// SIMATIC S7-200 project (STEP 7-Micro/WIN), CPU 224 REL 02.01

ORGANIZATION_BLOCK Briquette_Press_B_40:OB1
TITLE=B V4.0
// Custom program for WEIMA TH Standard Series briquette press.
//  #NVJOB Nicholas Veselov (independent developer) - https://nvjob.pro, http://nvjob.dx.am
// 
// ---------------------------------------------------------------------
// 
// INPUTS
// I0.0 - Power.
// I0.1 - Start the program in automatic mode.
// I0.2 - Stop the program in automatic mode.
// I0.3 - Manual mode.
// I0.4 - Vertical piston, sensor, lower position.
// I0.5 - Vertical piston, sensor, upper position.
// I0.6 - Horizontal piston, sensor, position retracted.
// I0.7 - Horizontal piston, sensor, position extended.
// I1.0 - Not involved.
// I1.1 - Valve button.
// I1.2 - Accident, stop.
// I1.3 - Change in operating time of the screw. Min time*.
// I1.4 - Change in the operating time of the screw. Max. time*.
// I1.5 - Not involved.
// 
// ---------------------------------------------------------------------
// 
// OUTPUTS
// Q0.0 - The engine of the hydraulic power station (star-delta).
// Q0.1 - Hydroelectric power station engine (star-delta).
// Q0.2 - Fan.
// Q0.3 - Auger.
// Q0.4 - Vertical piston, valve, up position (pushes down).
// Q0.5 - Vertical piston, valve, lower position (pushes up).
// Q0.6 - Horizontal piston, valve, retracts the piston.
// Q0.7 - Horizontal piston, valve, extends the piston.
// Q1.0 - Collet Piston.
// Q1.1 - Light Bulb Start
// 
BEGIN
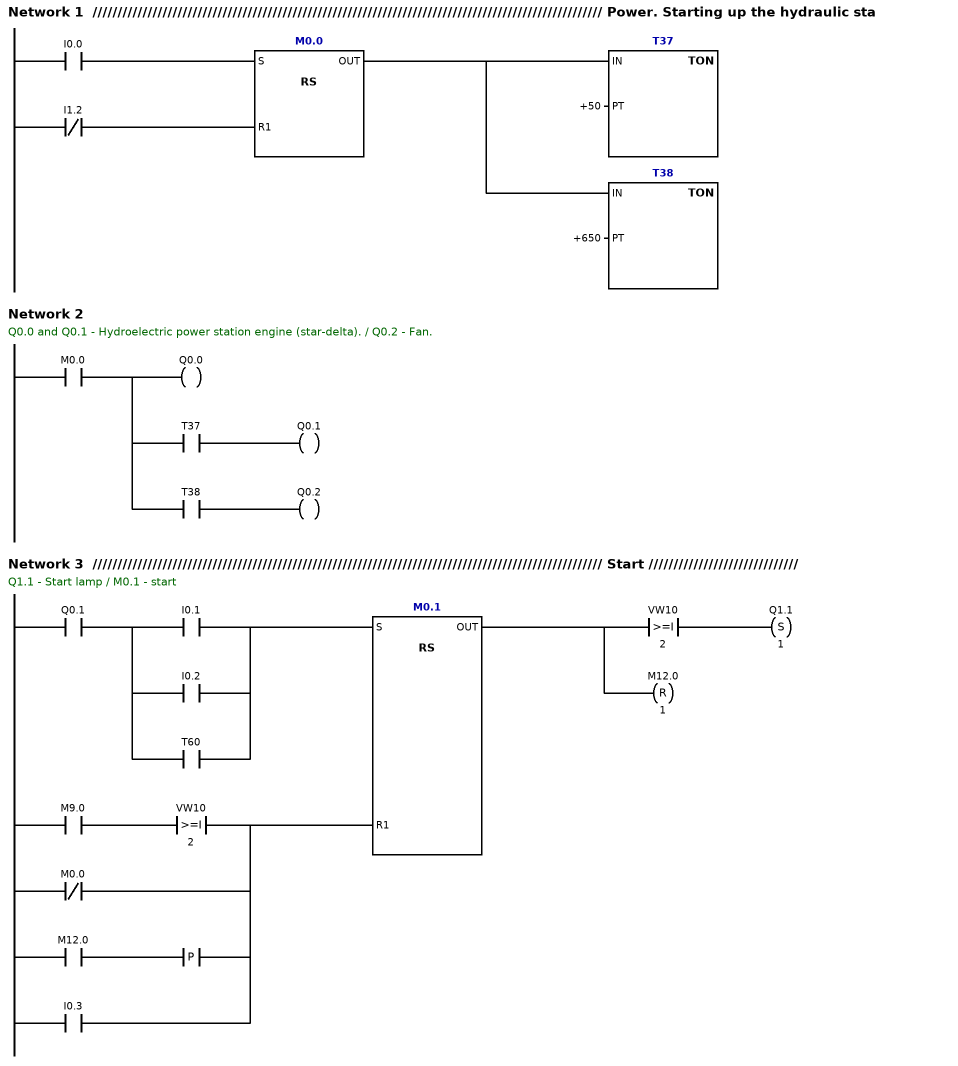
Network 1 // //////////////////////////////////////////////////////////////////////////////////////////////////////
Power. Starting up the hydraulic station.
//////////////////////////////////////////////////////////////////////////////////////////////////////
LD     I0.0
LDN    I1.2
NOT
LPS
A      M0.0
=      M0.0
LPP
ALD
O      M0.0
=      M0.0
TON    T37, +50
TON    T38, +650
Network 2
// Q0.0 and Q0.1 - Hydroelectric power station engine (star-delta).
// Q0.2 - Fan.
LD     M0.0
LPS
=      Q0.0
A      T37
=      Q0.1
LPP
A      T38
=      Q0.2
Network 3 // //////////////////////////////////////////////////////////////////////////////////////////////////////
Start
//////////////////////////////////////////////////////////////////////////////////////////////////////
// Q1.1 - Start lamp
// M0.1 - start
LD     Q0.1
LD     I0.1
O      I0.2
O      T60
ALD
LD     M9.0
AW>=   VW10, 2
ON     M0.0
LD     M12.0
EU
OLD
O      I0.3
NOT
LPS
A      M0.1
=      M0.1
LPP
ALD
O      M0.1
=      M0.1
LPS
AW>=   VW10, 2
S      Q1.1, 1
LPP
R      M12.0, 1
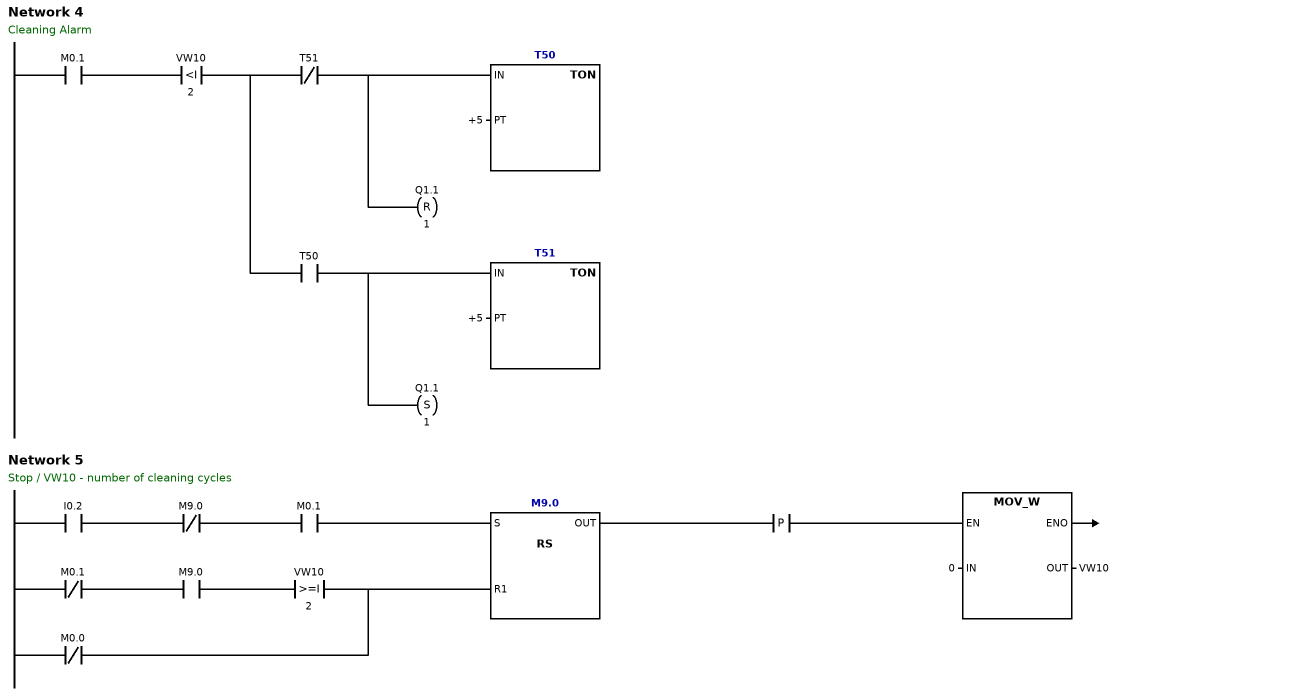
Network 4
// Cleaning Alarm
LD     M0.1
AW<    VW10, 2
LPS
AN     T51
TON    T50, +5
R      Q1.1, 1
LPP
A      T50
TON    T51, +5
S      Q1.1, 1
Network 5
// Stop
// VW10 - number of cleaning cycles
LD     I0.2
AN     M9.0
A      M0.1
LDN    M0.1
A      M9.0
AW>=   VW10, 2
ON     M0.0
NOT
LPS
A      M9.0
=      M9.0
LPP
ALD
O      M9.0
=      M9.0
EU
MOVW   0, VW10
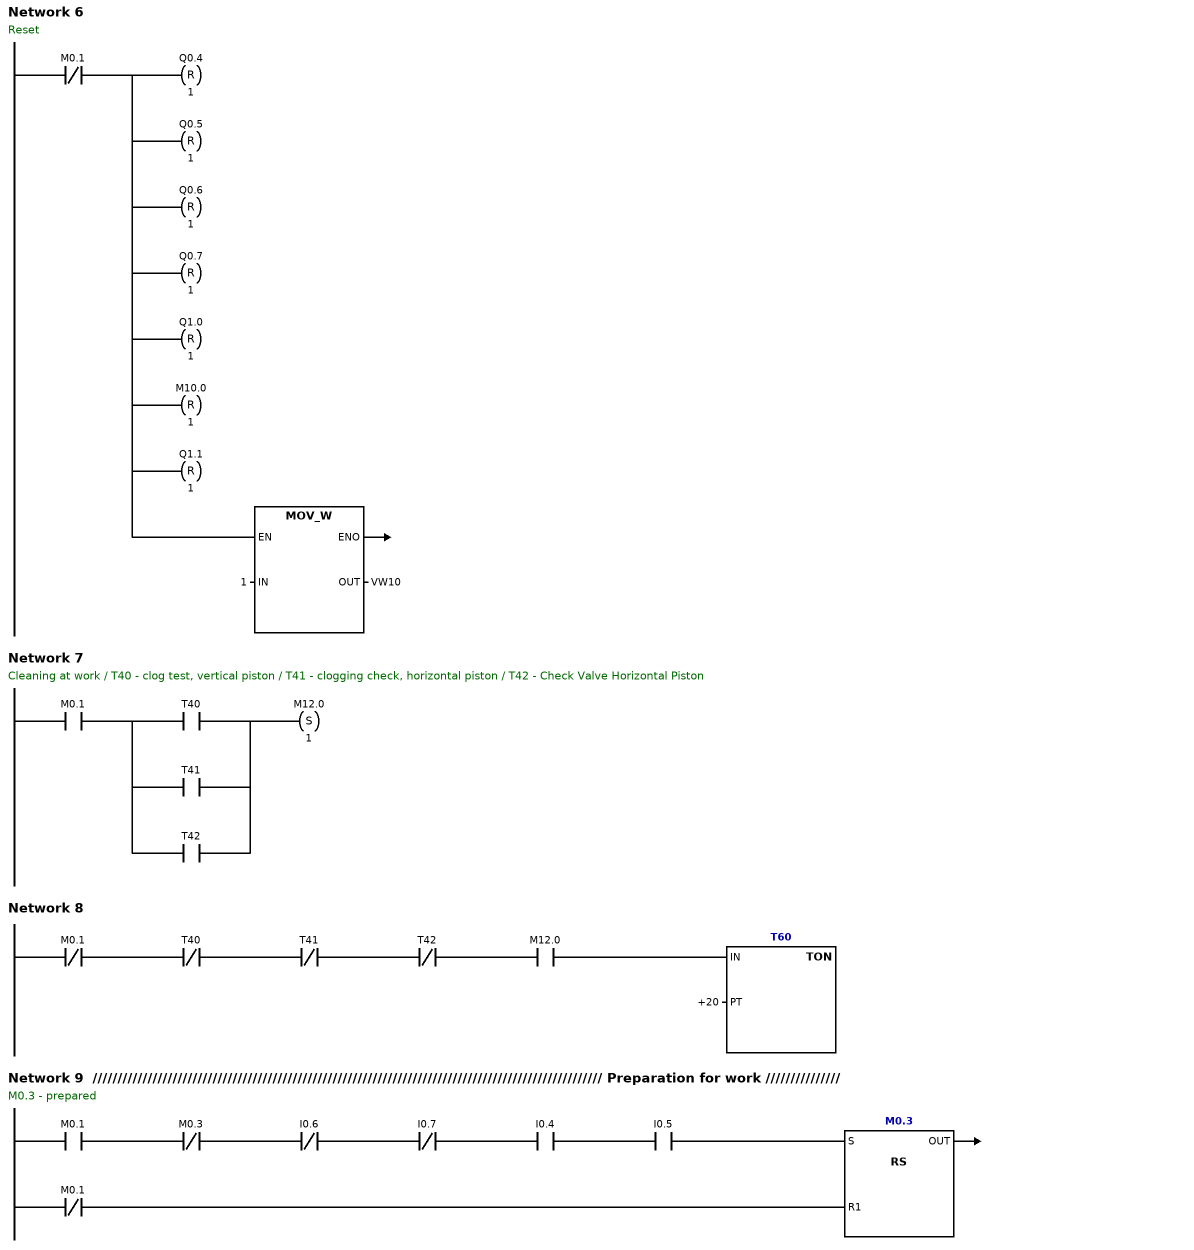
Network 6
// Reset
LDN    M0.1
R      Q0.4, 1
R      Q0.5, 1
R      Q0.6, 1
R      Q0.7, 1
R      Q1.0, 1
R      M10.0, 1
R      Q1.1, 1
MOVW   1, VW10
Network 7
// Cleaning at work
// T40 - clog test, vertical piston
// T41 - clogging check, horizontal piston
// T42 - Check Valve Horizontal Piston
LD     M0.1
LD     T40
O      T41
O      T42
ALD
S      M12.0, 1
Network 8
LDN    M0.1
AN     T40
AN     T41
AN     T42
A      M12.0
TON    T60, +20
Network 9 // //////////////////////////////////////////////////////////////////////////////////////////////////////
Preparation for work
//////////////////////////////////////////////////////////////////////////////////////////////////////
// M0.3 - prepared
LD     M0.1
AN     M0.3
AN     I0.6
AN     I0.7
A      I0.4
A      I0.5
LDN    M0.1
NOT
LPS
A      M0.3
=      M0.3
LPP
ALD
O      M0.3
=      M0.3
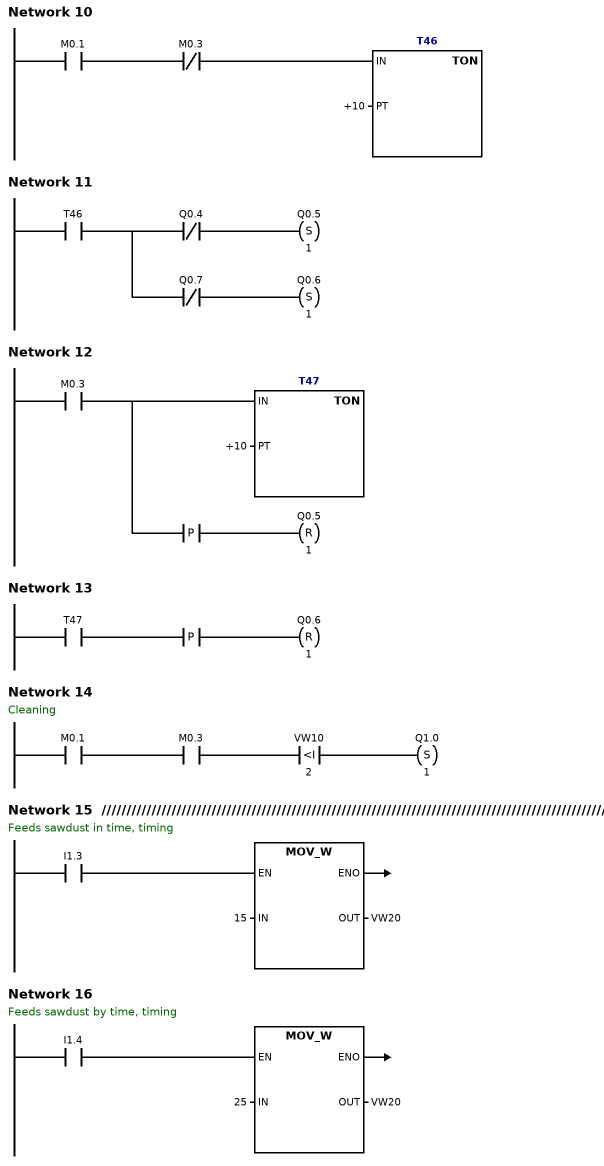
Network 10
LD     M0.1
AN     M0.3
TON    T46, +10
Network 11
LD     T46
LPS
AN     Q0.4
S      Q0.5, 1
LPP
AN     Q0.7
S      Q0.6, 1
Network 12
LD     M0.3
TON    T47, +10
EU
R      Q0.5, 1
Network 13
LD     T47
EU
R      Q0.6, 1
Network 14
// Cleaning
LD     M0.1
A      M0.3
AW<    VW10, 2
S      Q1.0, 1
Network 15 // //////////////////////////////////////////////////////////////////////////////////////////////////////
Work
//////////////////////////////////////////////////////////////////////////////////////////////////////
// Feeds sawdust in time, timing
LD     I1.3
MOVW   15, VW20
Network 16
// Feeds sawdust by time, timing
LD     I1.4
MOVW   25, VW20
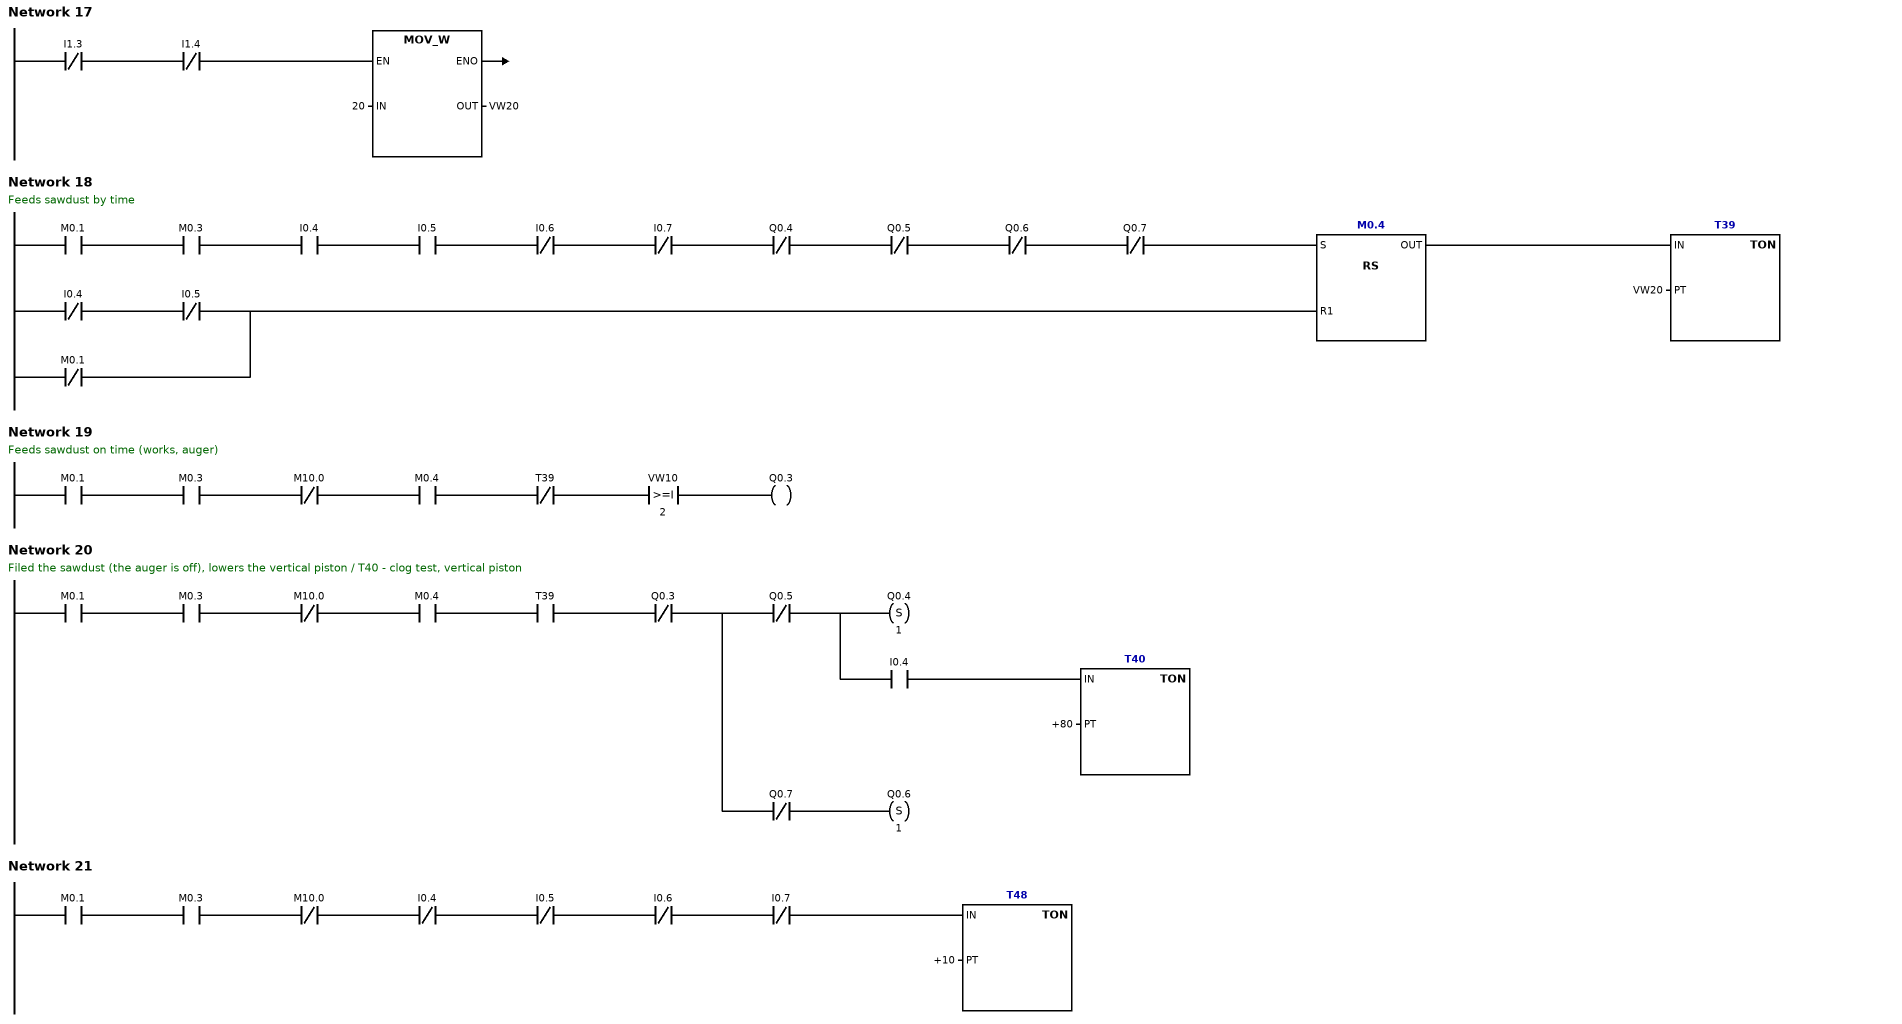
Network 17
LDN    I1.3
AN     I1.4
MOVW   20, VW20
Network 18
// Feeds sawdust by time
LD     M0.1
A      M0.3
A      I0.4
A      I0.5
AN     I0.6
AN     I0.7
AN     Q0.4
AN     Q0.5
AN     Q0.6
AN     Q0.7
LDN    I0.4
AN     I0.5
ON     M0.1
NOT
LPS
A      M0.4
=      M0.4
LPP
ALD
O      M0.4
=      M0.4
TON    T39, VW20
Network 19
// Feeds sawdust on time (works, auger)
LD     M0.1
A      M0.3
AN     M10.0
A      M0.4
AN     T39
AW>=   VW10, 2
=      Q0.3
Network 20
// Filed the sawdust (the auger is off), lowers the vertical piston
// T40 - clog test, vertical piston
LD     M0.1
A      M0.3
AN     M10.0
A      M0.4
A      T39
AN     Q0.3
LPS
AN     Q0.5
S      Q0.4, 1
A      I0.4
TON    T40, +80
LPP
AN     Q0.7
S      Q0.6, 1
Network 21
LD     M0.1
A      M0.3
AN     M10.0
AN     I0.4
AN     I0.5
AN     I0.6
AN     I0.7
TON    T48, +10
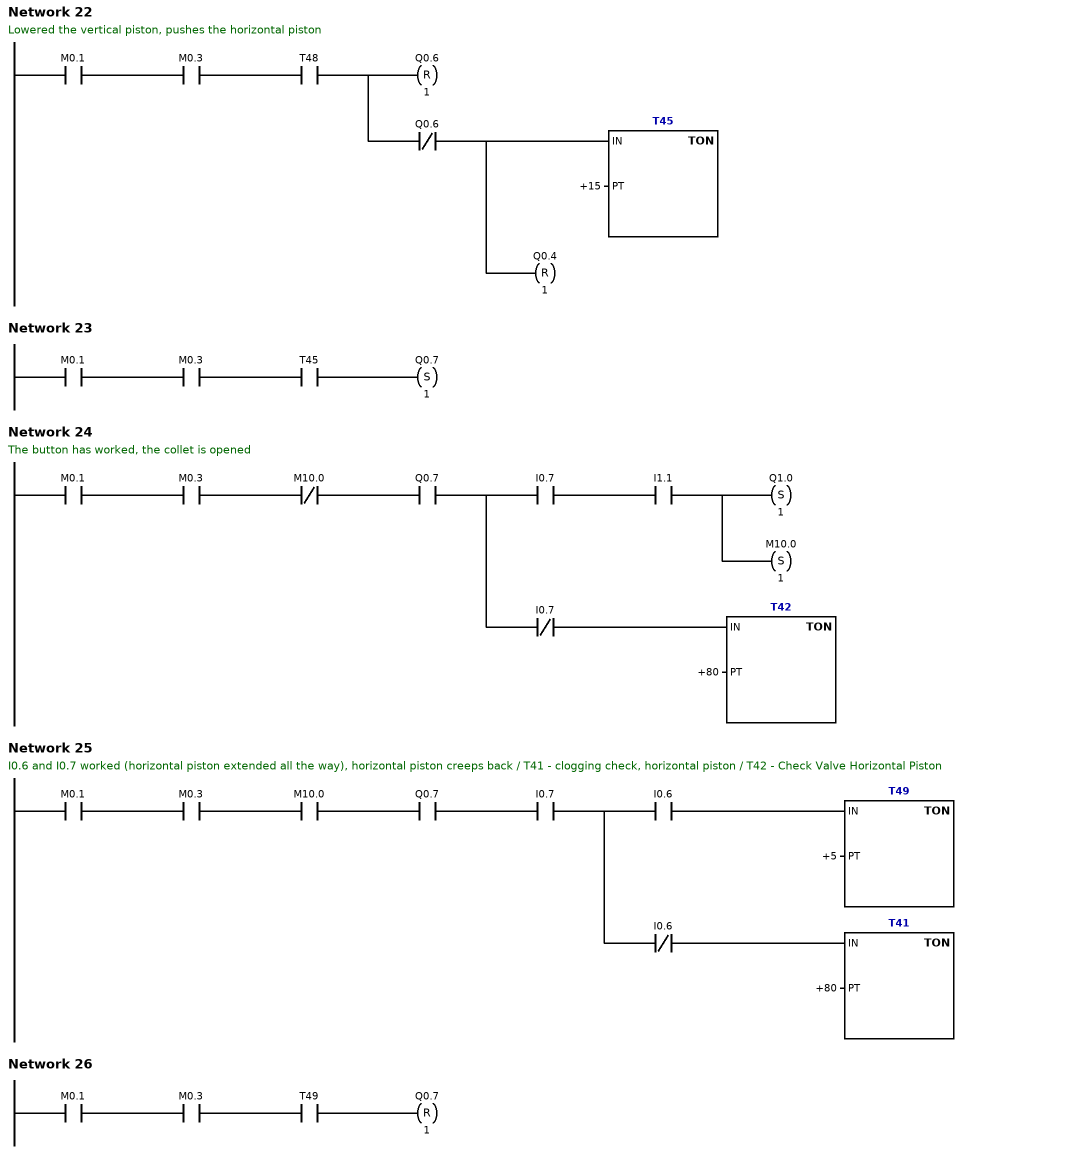
Network 22
// Lowered the vertical piston, pushes the horizontal piston
LD     M0.1
A      M0.3
A      T48
R      Q0.6, 1
AN     Q0.6
TON    T45, +15
R      Q0.4, 1
Network 23
LD     M0.1
A      M0.3
A      T45
S      Q0.7, 1
Network 24
// The button has worked, the collet is opened
LD     M0.1
A      M0.3
AN     M10.0
A      Q0.7
LPS
A      I0.7
A      I1.1
S      Q1.0, 1
S      M10.0, 1
LPP
AN     I0.7
TON    T42, +80
Network 25
// I0.6 and I0.7 worked (horizontal piston extended all the way), horizontal piston creeps back
// T41 - clogging check, horizontal piston
// T42 - Check Valve Horizontal Piston
LD     M0.1
A      M0.3
A      M10.0
A      Q0.7
A      I0.7
LPS
A      I0.6
TON    T49, +5
LPP
AN     I0.6
TON    T41, +80
Network 26
LD     M0.1
A      M0.3
A      T49
R      Q0.7, 1
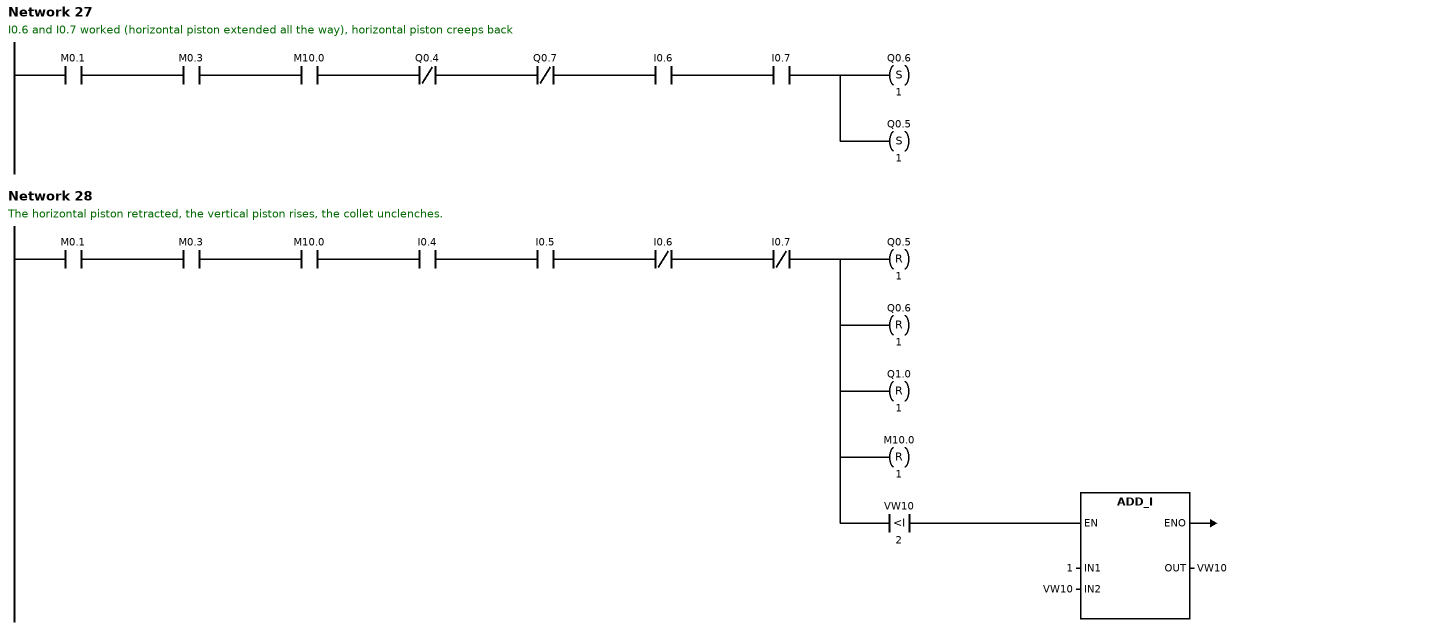
Network 27
// I0.6 and I0.7 worked (horizontal piston extended all the way), horizontal piston creeps back
LD     M0.1
A      M0.3
A      M10.0
AN     Q0.4
AN     Q0.7
A      I0.6
A      I0.7
S      Q0.6, 1
S      Q0.5, 1
Network 28
// The horizontal piston retracted, the vertical piston rises, the collet unclenches.
LD     M0.1
A      M0.3
A      M10.0
A      I0.4
A      I0.5
AN     I0.6
AN     I0.7
R      Q0.5, 1
R      Q0.6, 1
R      Q1.0, 1
R      M10.0, 1
AW<    VW10, 2
+I     1, VW10
END_ORGANIZATION_BLOCK
